% RSLogix 500 project PRELAB 3 CODE INT.RSS, saved by version 8.40.00.08 %
PROJECT "UNTITLED"    % processor: MicroLogix 1400 %

PROGRAM FILES
  LAD 2   12 rungs

DATA FILES
  O0 OUTPUT  6 elements
  I1 INPUT  8 elements
  S2 STATUS  66 elements
  B3 BINARY  1 elements
  T4 TIMER  3 elements
  C5 COUNTER  1 elements
  R6 CONTROL  1 elements
  N7 INTEGER  1 elements
  F8 FLOAT  1 elements

LADDER 2
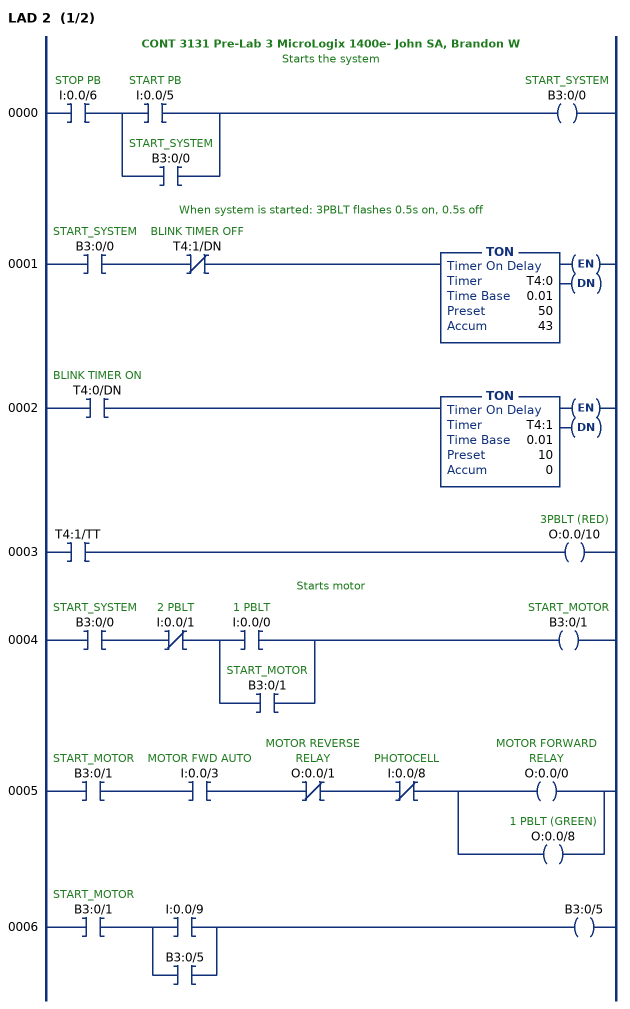
% Rung: 0 %
% TITLE: CONT 3131 Pre-Lab 3 MicroLogix 1400e- John SA, Brandon W %
% Starts the system %
SOR XIC I:0.0/6 BST XIC I:0.0/5 NXB XIC B3:0/0 BND OTE B3:0/0 EOR
%   I:0.0/6  "STOP PB" %
%   I:0.0/5  "START PB" %
%   B3:0/0  START_SYSTEM %
% Rung: 1 %
% When system is started: 3PBLT flashes 0.5s on, 0.5s off %
SOR XIC B3:0/0 XIO T4:1/DN TON T4:0 0.01 50 43 EOR
%   B3:0/0  START_SYSTEM %
%   T4:1/DN  "BLINK TIMER OFF" %
% Rung: 2 %
SOR XIC T4:0/DN TON T4:1 0.01 10 0 EOR
%   T4:0/DN  "BLINK TIMER ON" %
% Rung: 3 %
SOR XIC T4:1/TT OTE O:0.0/10 EOR
%   O:0.0/10  "3PBLT (RED)" %
% Rung: 4 %
% Starts motor %
SOR XIC B3:0/0 XIO I:0.0/1 BST XIC I:0.0/0 NXB XIC B3:0/1 BND OTE B3:0/1 EOR
%   B3:0/0  START_SYSTEM %
%   I:0.0/1  "2 PBLT" %
%   I:0.0/0  "1 PBLT" %
%   B3:0/1  START_MOTOR %
% Rung: 5 %
SOR XIC B3:0/1 XIC I:0.0/3 XIO O:0.0/1 XIO I:0.0/8 BST OTE O:0.0/0 NXB OTE O:0.0/8 BND EOR
%   B3:0/1  START_MOTOR %
%   I:0.0/3  "MOTOR FWD AUTO" %
%   O:0.0/1  "MOTOR REVERSE RELAY" %
%   I:0.0/8  "PHOTOCELL" %
%   O:0.0/0  "MOTOR FORWARD RELAY" %
%   O:0.0/8  "1 PBLT (GREEN)" %
% Rung: 6 %  % edit flag set %
SOR XIC B3:0/1 BST XIC I:0.0/9 NXB XIC B3:0/5 BND OTE B3:0/5 EOR
%   B3:0/1  START_MOTOR %

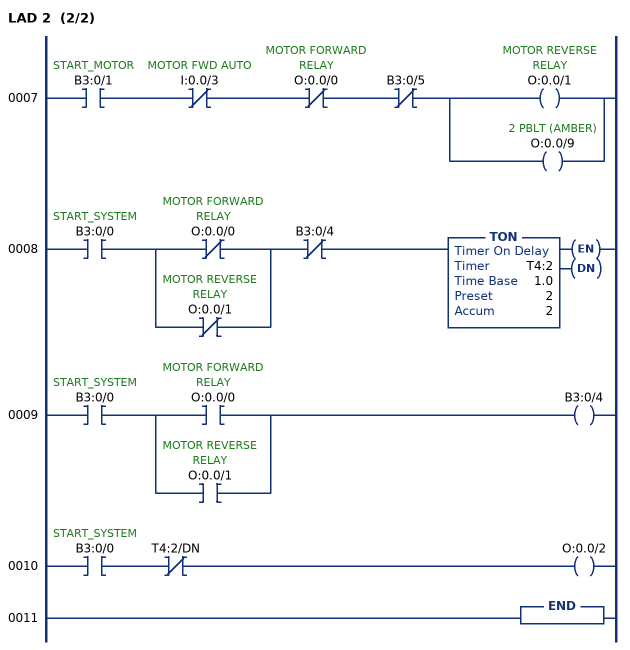
% Rung: 7 %  % edit flag set %
SOR XIC B3:0/1 XIO I:0.0/3 XIO O:0.0/0 XIO B3:0/5 BST OTE O:0.0/1 NXB OTE O:0.0/9 BND EOR
%   B3:0/1  START_MOTOR %
%   I:0.0/3  "MOTOR FWD AUTO" %
%   O:0.0/0  "MOTOR FORWARD RELAY" %
%   O:0.0/1  "MOTOR REVERSE RELAY" %
%   O:0.0/9  "2 PBLT (AMBER)" %
% Rung: 8 %
SOR XIC B3:0/0 BST XIO O:0.0/0 NXB XIO O:0.0/1 BND XIO B3:0/4 TON T4:2 1.0 2 2 EOR
%   B3:0/0  START_SYSTEM %
%   O:0.0/0  "MOTOR FORWARD RELAY" %
%   O:0.0/1  "MOTOR REVERSE RELAY" %
% Rung: 9 %
SOR XIC B3:0/0 BST XIC O:0.0/0 NXB XIC O:0.0/1 BND OTE B3:0/4 EOR
%   B3:0/0  START_SYSTEM %
%   O:0.0/0  "MOTOR FORWARD RELAY" %
%   O:0.0/1  "MOTOR REVERSE RELAY" %
% Rung: 10 %
SOR XIC B3:0/0 XIO T4:2/DN OTE O:0.0/2 EOR
%   B3:0/0  START_SYSTEM %
% Rung: 11 %
SOR END EOR

OTHER DOCUMENTED ADDRESSES
  I:1.0/0  1PBLT
  I:1.0/1  2PBLT
  I:1.0/3  FWD_REV
  I:1.0/5  START_PB
  I:1.0/6  STOP_PB
  I:1.0/8  PHOTOCELL
  I:1.0/9  LIMIT_SWITCH
  O:1.0/0  FWD_MOTOR
  O:1.0/1  REV_MOTOR
  O:1.0/8  1PBLT_LIGHT
  O:1.0/9  2PBLT_LIGHT
  O:1.0/10  3PBLT_LIGHT
  T1:0/DN  BLINK_TIMER
  T1:1/DN  MOTOR_OFF_DELAY

COMMENTS NOT ATTACHED TO A CURRENT RUNG
  O:1.0/3: Dynamic brake is active if both motor directions are de-activated
  T1:1: Shunt powers off if motor is active for 10 sec
  O:1.0/9: Reverse motor with limit switch
  O:1.0/8: Forward motor with photocell stop
  T1:0: Flashes red light

DATA TABLE (non-zero values as saved)
DATA B3
% B3:0 % 0X0001
DATA T4
% .PRE .ACC %
% T4:0 % 50 43
% T4:1 % 10 0
% T4:2 % 2 2
